INTERFACE ITF_LinkedList_Node EXTENDS __SYSTEM.IQueryInterface

PROPERTY p_IsLinkMaster : BOOL
GET
END_GET
END_PROPERTY

PROPERTY p_ListNext : ITF_LinkedList_Node
GET
END_GET
SET
END_SET
END_PROPERTY

PROPERTY p_ListPrevious : ITF_LinkedList_Node
GET
END_GET
SET
END_SET
END_PROPERTY

END_INTERFACE

(* stored: Version 1.1.0.1, ProductVersion 3.1.4024.12
   Itf ITF_LinkedList_Node: Id {9e732ef4-819a-4a28-bc73-2f3c564f0e55}
   Property p_IsLinkMaster: Id {6ba6d3a8-c654-4953-adcf-028da2ff855f}
   Get Get: Id {be4c69b2-31c6-488e-bcd4-1be63f64b77e}
   Property p_ListNext: Id {c7aacd18-7e8d-4845-a068-5a5b4c61cb1f}
   Get Get: Id {30060319-adfc-4b22-8a56-170135afd4fb}
   Set Set: Id {8075ab13-a6cb-4a8c-8a3e-1c61c6ee1240}
   Property p_ListPrevious: Id {96c8da52-abd8-4595-b354-8a66255646b8}
   Get Get: Id {e45a4399-f29e-4fa6-b3e2-1bc1faec3af7}
   Set Set: Id {add75c6e-3855-43cc-8a87-4869de2f681e} *)
